# EPICS alarm handler configuration: mps_database/bareTest/alarms/areas/mpln_bc1b_mp03.alhConfig
GROUP NULL MPLN:BC1B:MP03:1
$ALIAS MPS Link Node 59
$GUIDANCE
LTUH MPS
   Group Name: MPLN:BC1B:MP03:1
   Summary PV:  MPLN:BC1B:MP03:1:STATSUMY
$END
CHANNEL  MPLN:BC1B:MP03:1    MPLN:BC1B:MP03:1:MPS_EN_RBV		-----
CHANNEL  MPLN:BC1B:MP03:1    MPLN:BC1B:MP03:1:LC1_MODE_RBV		-----
